INTERFACE ITcoRestorable EXTENDS __SYSTEM.IQueryInterface

METHOD Restore : ITcoRestorable
END_METHOD

END_INTERFACE

(* stored: Version 1.1.0.1
   Itf ITcoRestorable: Id {62b2753f-f5a1-4b95-bc70-d5bc1062507d}
   Method Restore: Id {e2a78908-9be5-4407-99a7-5c57f7b6a6c9} *)
